(* PLC project contactor_2dir_1speed, Dassault Systèmes ControlBuild 2024x *)
(* stored: creationDateTime 2023-10-03T11:13:13-01:00 *)

(* This module simulates control system of motor. This motor has two directions and one speed. This system is represented by two contactors. *)
FUNCTION_BLOCK equipment_library.contactor_2dir_1speed
  VAR_INPUT
    voltage380 : BOOL := true;
    cmdSupply : BOOL := true;
    sensorSupply : BOOL := true;
  END_VAR
  VAR_INPUT
    forward : BOOL := false;
    backward : BOOL := false;
  END_VAR
  VAR_OUTPUT
    fwdHsState : BOOL := false;
    bwdHsState : BOOL := false;
  END_VAR
  VAR_OUTPUT
    forwardFB : BOOL := false;
    backwardFB : BOOL := false;
    thermal : BOOL := false;
  END_VAR
  VAR
    memoFwd : BOOL := false;
    memoBwd : BOOL := false;
  END_VAR
  VAR CONSTANT
    fwdLogic : BOOL := true;
    bwdLogic : BOOL := true;
    thermalLogic : BOOL := false;
  END_VAR
  VAR
    d_electrical : BOOL := false;
    v_d_electrical : BOOL := true;
    d_Bwd : BOOL := false;
    v_d_Bwd : BOOL := false;
    d_Fwd : BOOL := false;
    v_d_Fwd : BOOL := false;
  END_VAR


ACTION C_source_code:
/* ----------------------------------------------------------------	*/
/* Type : Model of Operative Behaviour					*/
/* Category :  Pre-actuators						*/
/* Author : Dassault Systemes						*/
/* Update date : June 2018							*/
/* ----------------------------------------------------------------	*/
/* This module simulates control system of motor. 			*/
/* This motor has two directions and one speed. 			*/
/* This system is represented by two contactors. 			*/
/* It returns its state and sensors' feed-back.				*/
/* ----------------------------------------------------------------	*/

/* ----------------------------------------------------------------	*/
/* Management of orders from Control Part					*/
/*	if there is no power supply for command 				*/
/*         the contactor doesn't understand the control orders.	*/
/* Contactors can't be actuated at the same time.			*/
/* Security is mchanical.							*/
/* ----------------------------------------------------------------	*/

memoFwd = forward && !memoBwd && cmdSupply && !d_electrical ;
memoBwd = backward && !memoFwd && cmdSupply && !d_electrical ;


/* ----------------------------------------------------------------	*/
/* Calculation of the on-state of contactors				*/
/* ----------------------------------------------------------------	*/
fwdHsState=memoFwd & voltage380;
bwdHsState=memoBwd & voltage380;

/* ----------------------------------------------------------------	*/
/* Management of the thermal feed-back					*/
/* ----------------------------------------------------------------	*/
if (d_electrical) thermal=v_d_electrical;
else
	thermal= ! thermalLogic && sensorSupply;

/* ----------------------------------------------------------------	*/
/* Management of feedback to Control Part					*/
/*     if a fault is required, the contactor feed-back 		*/
/*		 takes a preset state.					*/
/*	if there is no power supply for sensor 				*/
/*         contactor feed-back returns nothing				*/
/*     else contactor feed-back returns the contactor state combined	*/
/*	    with wiring logic.						*/
/* ----------------------------------------------------------------	*/
if (d_Fwd) forwardFB=v_d_Fwd;
else
	forwardFB=(memoFwd ^ ! fwdLogic) && sensorSupply;

if (d_Bwd) backwardFB=v_d_Bwd;
else
	backwardFB=(memoBwd ^ ! bwdLogic) && sensorSupply;
END_ACTION
END_FUNCTION_BLOCK
